TYPE ST_IOInputSimul :
STRUCT
	IxAru :BOOL;
END_STRUCT
END_TYPE

(* stored: Version 1.1.0.1, ProductVersion 3.1.4020.6
   DUT ST_IOInputSimul: Id {d975d12d-7e8d-4225-b1f2-f54f3150cc91} *)
